// Mitsubishi GX Works2 project: ZP.PSTRT 함수 동작 테스트   PLC: Q03UDV

PROGRAM MAIN
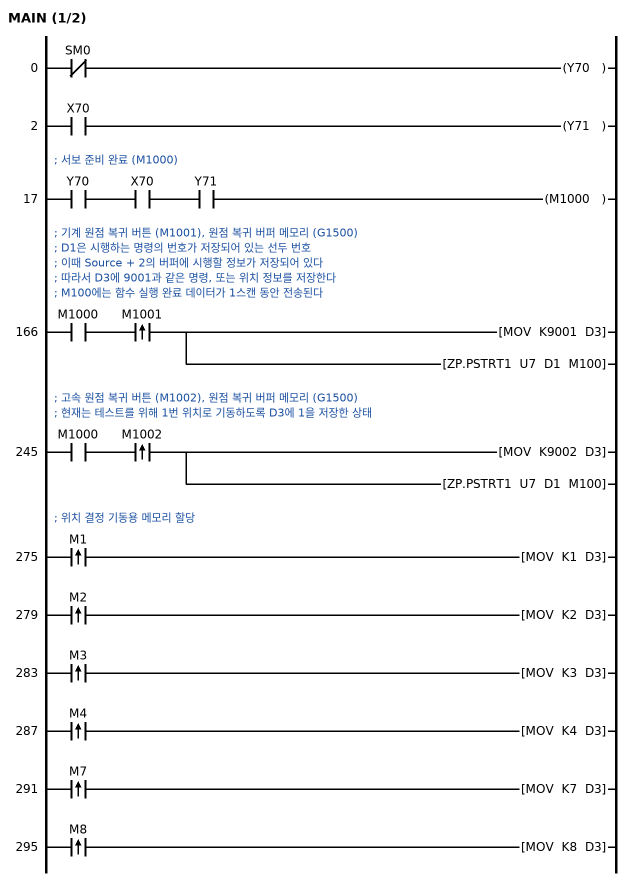
0     LDI     SM0
      OUT     Y70
2     LD      X70
      OUT     Y71
; 서보 준비 완료 (M1000)
17    LD      Y70
      AND     X70
      AND     Y71
      OUT     M1000
; 기계 원점 복귀 버튼 (M1001), 원점 복귀 버퍼 메모리 (G1500)
; D1은 시행하는 명령의 번호가 저장되어 있는 선두 번호
; 이때 Source + 2의 버퍼에 시행할 정보가 저장되어 있다
; 따라서 D3에 9001과 같은 명령, 또는 위치 정보를 저장한다
; M100에는 함수 실행 완료 데이터가 1스캔 동안 전송된다
166   LD      M1000
      ANDP    M1001
      MOV     K9001 D3
      ZP.PSTRT1 U7 D1 M100
; 고속 원점 복귀 버튼 (M1002), 원점 복귀 버퍼 메모리 (G1500)
; 현재는 테스트를 위해 1번 위치로 기동하도록 D3에 1을 저장한 상태
245   LD      M1000
      ANDP    M1002
      MOV     K9002 D3
      ZP.PSTRT1 U7 D1 M100
; 위치 결정 기동용 메모리 할당
275   LDP     M1
      MOV     K1 D3
279   LDP     M2
      MOV     K2 D3
283   LDP     M3
      MOV     K3 D3
287   LDP     M4
      MOV     K4 D3
291   LDP     M7
      MOV     K7 D3
295   LDP     M8
      MOV     K8 D3
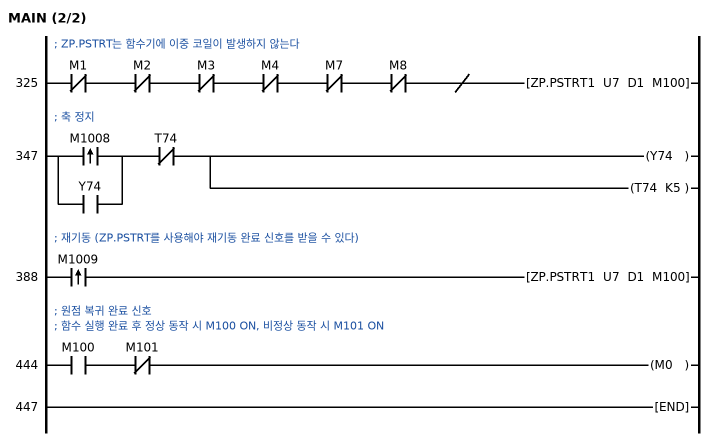
; ZP.PSTRT는 함수기에 이중 코일이 발생하지 않는다
325   LDI     M1
      ANI     M2
      ANI     M3
      ANI     M4
      ANI     M7
      ANI     M8
      INV
      ZP.PSTRT1 U7 D1 M100
; 축 정지
347   LDP     M1008
      OR      Y74
      ANI     T74
      OUT     Y74
      OUT     T74 K5
; 재기동 (ZP.PSTRT를 사용해야 재기동 완료 신호를 받을 수 있다)
388   LDP     M1009
      ZP.PSTRT1 U7 D1 M100
; 원점 복귀 완료 신호
; 함수 실행 완료 후 정상 동작 시 M100 ON, 비정상 동작 시 M101 ON
444   LD      M100
      ANI     M101
      OUT     M0
447   END
END_PROGRAM
